{attribute addProperty BoxType "EJ6224-0000-0016"}
{attribute addProperty Id "DeviceState_Inputs_DeviceDeviceState_Inputs_Device_345DC0EE162"}
{attribute addProperty CRC "1356676245"}
{attribute addProperty SizeInBites "16"}
{attribute addProperty SizeInBytes "2"}
TYPE Module_1_DeviceState_Inputs_Device_50DD3C95 :
STRUCT
	{attribute addProperty Name "DeviceState_Inputs_Device"}
	DeviceState_Inputs_Device  : DeviceState_Inputs_Device_345DC0EE;
END_STRUCT
END_TYPE

(* stored: Version 1.2.0.0, ProductVersion 3.1.4024.9
   DUT Module_1_DeviceState_Inputs_Device_50DD3C95: Id {6f4a87db-205a-4e62-a179-30ad501aa5d7} *)
